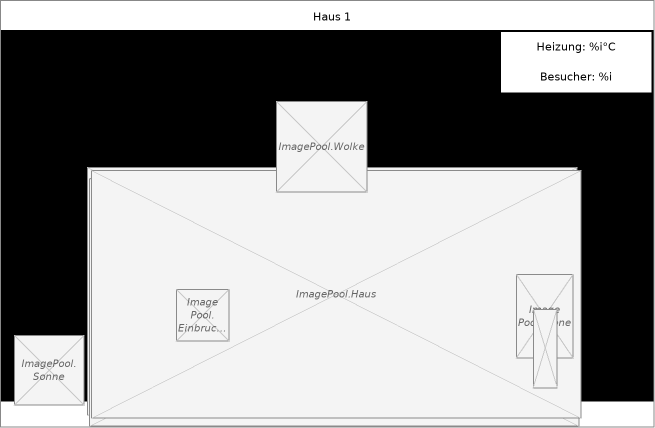
VISUALIZATION Haus_1  // 655x428
    Rectangle (1,30 652x371)
    Rectangle (1,30 652x371), colour variable: L_Himmel
        p2167032090: L_Himmel
    Image (87,167 490x248), invisible if: NOT net_licht_01, image: ImagePool.Dunkel
    Image (89,178 490x248), invisible if: net_licht_01, image: ImagePool.Licht
    Image (91,170 490x248), image: ImagePool.Haus
    Image (516,274 57x84), image: ImagePool.Krone
        p2858320360: L_Baum
    Image (533,309 24x79), image: ImagePool.Stamm
    Image (14,335 70x70), image: ImagePool.Sonne
        p2858320360: L_Sonnenstand
        p84334746: L_Sonne
    Image (176,289 53x52), image: ImagePool.Einbruch_grun
        p84334746: Haus1.L_EinbruchBild
    Image (276,101 91x91), image: ImagePool.Wolke
        p84334746: Haus1.WetterBild
    Textfield (257,6 150x22), "Haus 1"
    Textfield (501,32 150x30), "Heizung: %i°C", text variable: net_heizung_01
    Textfield (501,62 150x30), "Besucher: %i", text variable: net_besucher_01
END_VISUALIZATION

(* stored: Version 1.1.0.1, ProductVersion 3.1.4018.5
   Visu Haus_1: Id {3a34ba57-b0ad-46e3-811d-5feae23b576c} *)
